FUNCTION_BLOCK AutomationControl_1
VAR_INPUT
	piston1for: BOOL;
	piston1back: BOOL;
	
	piston2for: BOOL;
	piston2back: BOOL;
	
	pistonVert: BOOL;
	
	motorRotate: BOOL;
	
	motorCon: BOOL;
	
END_VAR
VAR
	sleeping1: sleep;
	sleeping2: sleep;
END_VAR


//Piston1
GVL.Piston1For := piston1for;
GVL.Piston1Back := piston1back;

//Piston2
GVL.Piston2For := piston2for;
GVL.Piston2Back := piston2back;

GVL.PistonVert := pistonVert;

GVL.MotorCon := motorCon;

GVL.MotorRotate := motorRotate;

END_FUNCTION_BLOCK

(* stored: Version 1.1.0.1, ProductVersion 3.1.4024.12
   POU AutomationControl_1: Id {e7b10cb8-bfcc-4411-a441-ce2ad54738ab}, SpecialFunc None *)
